// TIA Portal V17 export
// export: Created 2024-08-20T13:36:58.9429337Z, ExportSetting WithDefaults, DisplayName Totally Integrated Automation Portal, DisplayVersion V17 Update 4, DisplayName TIA Portal Openness, DisplayVersion V17 Update 4, DisplayName TIA Portal Version Control Interface, DisplayVersion V17, DisplayName STEP 7 Professional, DisplayVersion V17 Update 4, DisplayName STEP 7 Safety, DisplayVersion V17, DisplayName WinCC Advanced, DisplayVersion V17 Update 4
FUNCTION_BLOCK "PDIR"   // FB207, LAD
{ S7_Optimized_Access := 'FALSE' }
VERSION : 0.1
// stored: AutoNumber false, IsIECCheckEnabled false, SetENOAutomatically false, UDAEnableTagReadback false
   VAR_INPUT
      ML : Bool;
      MR : Bool;
      DL : Bool;
      MF1 : Bool;
      MF2 : Bool;
      HM : Bool;
      HA : Bool;
      CMA : Bool;
      CLM : Bool;
      CDM : Bool;
      CRF : Bool;
      CRTO : Bool;
      CL1S : Bool;
   END_VAR
   VAR_OUTPUT
      YFPP : Bool;
      YF : Bool;
      CL : Bool;
   END_VAR
   VAR_IN_OUT
      SEG : Int;
      MIN : Int;
      HOR : Int;
   END_VAR
   VAR DB_SPECIFIC
      AUX01 : Bool;
      AUX02 : Bool;
      AUX03 : Bool;
      AUX04 : Bool;
      AUX05 : Bool;
      AUX06 : Bool;
      AUX07 : Bool;
      AUX08 : Bool;
      AUX09 : Bool;
      P60S : Bool;
      P60M : Bool;
      PFHO : Bool;
      TPP1 { S7_SetPoint := 'True'} : TON_TIME;
      TPP2 { S7_SetPoint := 'True'} : TON_TIME;
   END_VAR
   VAR_TEMP
      TEMP0 : Bool;
      TEMP1 : Bool;
      ET_TPP1 : Time;
      ET_TPP2 : Time;
   END_VAR
   VAR_TEMP   // added for the SCL form of the ladder/FBD networks
      _w1 : Bool;
      _w2 : Bool;
      _w3 : Bool;
      _w4 : Bool;
   END_VAR
BEGIN

REGION Network 1: Falha na partida
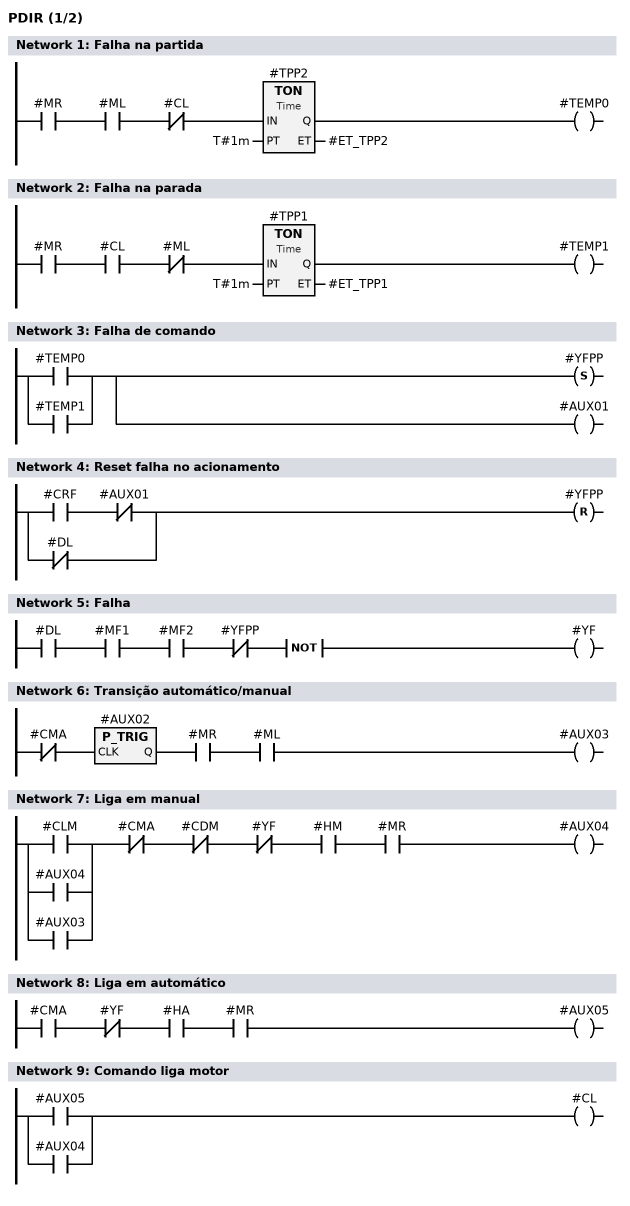
   RUNG wire#powerrail
      Contact( #MR )
      Contact( #ML )
      I_Contact( #CL )
      { S7_Templates := "time_type := Time" } #TPP2.TON(pt := T#1m, et => #ET_TPP2)
      Coil( #TEMP0 )
   END_RUNG
   // the same network as SCL:
   #TPP2(IN := #MR AND #ML AND NOT #CL, PT := T#1m, ET => #ET_TPP2);   // TON
   #TEMP0 := #TPP2.Q;
END_REGION

REGION Network 2: Falha na parada
   RUNG wire#powerrail
      Contact( #MR )
      Contact( #CL )
      I_Contact( #ML )
      { S7_Templates := "time_type := Time" } #TPP1.TON(pt := T#1m, et => #ET_TPP1)
      Coil( #TEMP1 )
   END_RUNG
   // the same network as SCL:
   #TPP1(IN := #MR AND #CL AND NOT #ML, PT := T#1m, ET => #ET_TPP1);   // TON
   #TEMP1 := #TPP1.Q;
END_REGION

REGION Network 3: Falha de comando
   RUNG wire#powerrail
      Contact( #TEMP0 )
      wire#w1
      S_Coil( #YFPP )
   END_RUNG
   RUNG wire#powerrail
      Contact( #TEMP1 )
   END_RUNG wire#w1
   RUNG wire#w1
      Coil( #AUX01 )
   END_RUNG
   // the same network as SCL:
   #_w1 := #TEMP0 OR #TEMP1;
   IF #_w1 THEN #YFPP := TRUE; END_IF;
   #AUX01 := #_w1;
END_REGION

REGION Network 4: Reset falha no acionamento
   RUNG wire#powerrail
      Contact( #CRF )
      I_Contact( #AUX01 )
      wire#w1
      R_Coil( #YFPP )
   END_RUNG
   RUNG wire#powerrail
      I_Contact( #DL )
   END_RUNG wire#w1
   // the same network as SCL:
   IF (#CRF AND NOT #AUX01) OR NOT #DL THEN #YFPP := FALSE; END_IF;
END_REGION

REGION Network 5: Falha
   RUNG wire#powerrail
      Contact( #DL )
      Contact( #MF1 )
      Contact( #MF2 )
      I_Contact( #YFPP )
      Not()
      Coil( #YF )
   END_RUNG
   // the same network as SCL:
   #YF := NOT (#DL AND #MF1 AND #MF2 AND NOT #YFPP);
END_REGION

REGION Network 6: Transição automático/manual
   RUNG wire#powerrail
      I_Contact( #CMA )
      P_Trig( #AUX02 )
      Contact( #MR )
      Contact( #ML )
      Coil( #AUX03 )
   END_RUNG
   // the same network as SCL:
   #_w1 := NOT #CMA AND NOT #AUX02;   // rising edge
   #AUX02 := NOT #CMA;
   #AUX03 := #_w1 AND #MR AND #ML;
END_REGION

REGION Network 7: Liga em manual
   RUNG wire#powerrail
      Contact( #CLM )
      wire#w1
      I_Contact( #CMA )
      I_Contact( #CDM )
      I_Contact( #YF )
      Contact( #HM )
      Contact( #MR )
      Coil( #AUX04 )
   END_RUNG
   RUNG wire#powerrail
      Contact( #AUX04 )
   END_RUNG wire#w1
   RUNG wire#powerrail
      Contact( #AUX03 )
   END_RUNG wire#w1
   // the same network as SCL:
   #AUX04 := (#CLM OR #AUX04 OR #AUX03) AND NOT #CMA AND NOT #CDM AND NOT #YF AND #HM AND #MR;
END_REGION

REGION Network 8: Liga em automático
   RUNG wire#powerrail
      Contact( #CMA )
      I_Contact( #YF )
      Contact( #HA )
      Contact( #MR )
      Coil( #AUX05 )
   END_RUNG
   // the same network as SCL:
   #AUX05 := #CMA AND NOT #YF AND #HA AND #MR;
END_REGION

REGION Network 9: Comando liga motor
   RUNG wire#powerrail
      Contact( #AUX05 )
      wire#w1
      Coil( #CL )
   END_RUNG
   RUNG wire#powerrail
      Contact( #AUX04 )
   END_RUNG wire#w1
   // the same network as SCL:
   #CL := #AUX05 OR #AUX04;
END_REGION

REGION Network 10
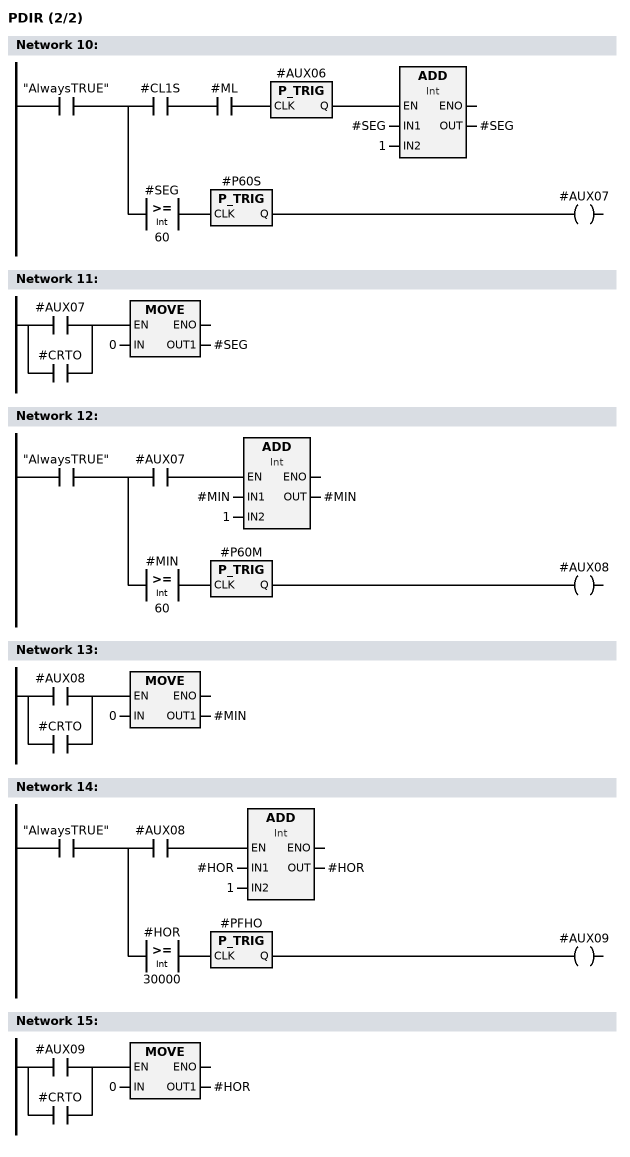
   RUNG wire#powerrail
      Contact( "AlwaysTRUE" )
      wire#w1
      Contact( #CL1S )
      Contact( #ML )
      P_Trig( #AUX06 )
      { S7_Templates := "SrcType := Int"; S7_GenerateENO := "TRUE" } Add(in1 := #SEG, in2 := 1, out => #SEG)
   END_RUNG
   RUNG wire#w1
      { S7_Templates := "SrcType := Int" } GE_Contact(in1 := #SEG, in2 := 60)
      P_Trig( #P60S )
      Coil( #AUX07 )
   END_RUNG
   // the same network as SCL:
   #_w1 := "AlwaysTRUE" AND #CL1S AND #ML;
   #_w2 := #_w1 AND NOT #AUX06;   // rising edge
   #AUX06 := #_w1;
   IF #_w2 THEN #SEG := #SEG + 1; END_IF;
   #_w3 := "AlwaysTRUE" AND (#SEG >= 60);
   #_w4 := #_w3 AND NOT #P60S;   // rising edge
   #P60S := #_w3;
   #AUX07 := #_w4;
END_REGION

REGION Network 11
   RUNG wire#powerrail
      Contact( #AUX07 )
      wire#w1
      { S7_GenerateENO := "TRUE" } Move(in := 0, out1 => #SEG)
   END_RUNG
   RUNG wire#powerrail
      Contact( #CRTO )
   END_RUNG wire#w1
   // the same network as SCL:
   IF #AUX07 OR #CRTO THEN #SEG := 0; END_IF;
END_REGION

REGION Network 12
   RUNG wire#powerrail
      Contact( "AlwaysTRUE" )
      wire#w1
      Contact( #AUX07 )
      { S7_Templates := "SrcType := Int"; S7_GenerateENO := "TRUE" } Add(in1 := #MIN, in2 := 1, out => #MIN)
   END_RUNG
   RUNG wire#w1
      { S7_Templates := "SrcType := Int" } GE_Contact(in1 := #MIN, in2 := 60)
      P_Trig( #P60M )
      Coil( #AUX08 )
   END_RUNG
   // the same network as SCL:
   IF "AlwaysTRUE" AND #AUX07 THEN #MIN := #MIN + 1; END_IF;
   #_w1 := "AlwaysTRUE" AND (#MIN >= 60);
   #_w2 := #_w1 AND NOT #P60M;   // rising edge
   #P60M := #_w1;
   #AUX08 := #_w2;
END_REGION

REGION Network 13
   RUNG wire#powerrail
      Contact( #AUX08 )
      wire#w1
      { S7_GenerateENO := "TRUE" } Move(in := 0, out1 => #MIN)
   END_RUNG
   RUNG wire#powerrail
      Contact( #CRTO )
   END_RUNG wire#w1
   // the same network as SCL:
   IF #AUX08 OR #CRTO THEN #MIN := 0; END_IF;
END_REGION

REGION Network 14
   RUNG wire#powerrail
      Contact( "AlwaysTRUE" )
      wire#w1
      Contact( #AUX08 )
      { S7_Templates := "SrcType := Int"; S7_GenerateENO := "TRUE" } Add(in1 := #HOR, in2 := 1, out => #HOR)
   END_RUNG
   RUNG wire#w1
      { S7_Templates := "SrcType := Int" } GE_Contact(in1 := #HOR, in2 := 30000)
      P_Trig( #PFHO )
      Coil( #AUX09 )
   END_RUNG
   // the same network as SCL:
   IF "AlwaysTRUE" AND #AUX08 THEN #HOR := #HOR + 1; END_IF;
   #_w1 := "AlwaysTRUE" AND (#HOR >= 30000);
   #_w2 := #_w1 AND NOT #PFHO;   // rising edge
   #PFHO := #_w1;
   #AUX09 := #_w2;
END_REGION

REGION Network 15
   RUNG wire#powerrail
      Contact( #AUX09 )
      wire#w1
      { S7_GenerateENO := "TRUE" } Move(in := 0, out1 => #HOR)
   END_RUNG
   RUNG wire#powerrail
      Contact( #CRTO )
   END_RUNG wire#w1
   // the same network as SCL:
   IF #AUX09 OR #CRTO THEN #HOR := 0; END_IF;
END_REGION
END_FUNCTION_BLOCK
